// TwinCAT 3 PLC project MCSB
// ProgramVersion: 3.1.4024.0
// libraries:
//   Tc2_MC2, * (Beckhoff Automation GmbH)
//   Tc2_MC2_Drive, * (Beckhoff Automation GmbH)
//   Tc2_Standard, * (Beckhoff Automation GmbH)
//   Tc2_System, * (Beckhoff Automation GmbH)
//   Tc2_Utilities, * (Beckhoff Automation GmbH)
//   Tc3_Module, * (Beckhoff Automation GmbH)
// project tree:
//   DUTs/ ST_MC_CMD.TcDUT, ST_MC_Status.TcDUT
//   GVLs/ GVL.TcGVL
//   / PlcTask.TcTTO
//   POUs/ MAIN.TcPOU, MotionCtrl.TcPOU
// real-time tasks:
//   TASK PlcTask: cycle T#10ms, priority 20, ADS port 350
// motion (NC):
//   TASK NC-Task 1 SAF: cycle T#2ms, priority 4, ADS port 501
//   TASK NC-Task 1 SVB: cycle T#10ms, priority 8, ADS port 511
//   AXIS Axis 1 (id 1)
//     OtherSettings: AllowMotionCmdToSlave=true
//     encoder EncType=19
//       EncPara: MaxCount=#xffffffff
//     drive DrvType=16
//       DrvPara: MaxCount=#xffffffff
//         Analog: TorqueSetpointScale=10, ScaleFactorActTorque=0.1
//         TimeComp: TaskDelayCycles=1
//     controller CtrType=1
//       CtrPara: PriorControlFactor=1
//         Observer: BandWidth=20
//   AXIS Axis 2 (id 2)
//     Dynamic: Acceleration=1610, Deceleration=1610, Jerk=2124.67
//     OtherSettings: AllowMotionCmdToSlave=true
//     encoder EncType=7
//       EncPara: MaxCount=#x0000ffff, ReferenceSystem=1
//     drive DrvType=5
//       Analog: TorqueSetpointScale=10, ScaleFactorActTorque=0.1
//       TimeComp: TaskDelayCycles=1
//     controller CtrType=1
//       CtrPara: PriorControlFactor=1
//         Observer: BandWidth=20
//   AXIS Axis 3 Virtual (id 3)
//     OtherSettings: AllowMotionCmdToSlave=true
//     encoder EncType=1
//     drive DrvType=5
//       Analog: TorqueSetpointScale=10, ScaleFactorActTorque=0.1
//       TimeComp: TaskDelayCycles=1
//     controller CtrType=1
//       CtrPara: PriorControlFactor=1
//         Observer: BandWidth=20
// I/O:
//   DEVICE Device 1 (EtherCAT) (disabled), AmsNetId 10.0.2.15.2.1
//     Term 1 (EK1200) [EK1200-5000 EtherCAT Power supply (2A E-Bus)]
//       Term 2 (EL1008) [EL1008 8Ch. Dig. Input 24V, 3ms]
//       Term 3 (EL2008) [EL2008 8Ch. Dig. Output 24V, 0.5A]
//       Drive 4 (EL7201-0001) [EL7201-0001 1Ch. DS402 Servo motor output stage (50V, 4A)]
//       Term 5 (EL3042) [EL3042 2Ch. Ana. Input 0-20mA]
//       Term 6 (EL4012) [EL4012 2Ch. Ana. Output 0-20mA, 12bit]
//       Term 7 (EK1122) [EK1122 2 port EtherCAT junction]
// variable links:
//   MCSB/MCSB Instance <-> NC-Task 1 SAF/Axes/Axis 3 Virtual
//     PlcTask Inputs/GVL.SingleAxis.NcToPlc <-> Outputs/ToPlc
//     PlcTask Outputs/GVL.SingleAxis.PlcToNc <-> Inputs/FromPlc
//   (this object) <-> Device 1 (EtherCAT)/Term 1 (EK1200)/Drive 4 (EL7201-0001)
//     Drive/Inputs/In/nDcOutputTime <-> InfoData/DcOutputShift
//     Drive/Inputs/In/nState1 <-> DS402 Statusword/Statusword
//     Drive/Inputs/In/nState2 <-> DS402 Statusword/Statusword @bit 8
//     Drive/Inputs/In/nState4 @bit 1 <-> WcState/InputToggle
//     Drive/Inputs/In/nState4 <-> WcState/WcState
//     Drive/Outputs/Out/nCtrl1 <-> DS402 Controlword/Controlword
//     Drive/Outputs/Out/nCtrl2 <-> DS402 Controlword/Controlword @bit 8
//     Drive/Outputs/Out/nDataOut2 <-> DS402 Target velocity/Target velocity
//     Enc/Inputs/In/nDataIn1 <-> DS402 Position actual value/Position actual value
//     Enc/Inputs/In/nDcInputTime <-> InfoData/DcInputShift
//     Enc/Inputs/In/nState4 @bit 1 <-> WcState/InputToggle
//     Enc/Inputs/In/nState4 <-> WcState/WcState
//   (this object) <-> Device 1 (EtherCAT)/Term 1 (EK1200)/Term 5 (EL3042)
//     Enc/Inputs/In/nDataIn1[0] <-> AI Standard Channel 1/Value
//     Enc/Inputs/In/nState4 @bit 1 <-> WcState/InputToggle
//     Enc/Inputs/In/nState4 <-> WcState/WcState
//   (this object) <-> Device 1 (EtherCAT)/Term 1 (EK1200)/Term 6 (EL4012)
//     Drive/Inputs/In/nState4 <-> WcState/WcState
//     Drive/Outputs/Out/nDataOut1[0] <-> AO Outputs Channel 1/Analog output

CONFIGURATION MCSB
    RESOURCE PLC ON TwinCAT3
        TASK PlcTask(INTERVAL := T#10ms, PRIORITY := 20);
        PROGRAM MAIN WITH PlcTask : MAIN;
    END_RESOURCE
END_CONFIGURATION

// ---- DUTs/ST_MC_CMD.TcDUT
TYPE ST_MC_CMD :
STRUCT
	bExe	  		: BOOL;
	lrVelocity		: LREAL;
	lrAcceleration	: LREAL;
	lrDeceleration	: LREAL;
	lrJog			: LREAL;
	lrDistance		: LREAL;
	lrPosition		: LREAL;
	EnuDrecetion	: MC_Direction;
	EnuBufferMode	: MC_BufferMode;
	EnuOptions		: ST_MoveOptions;
END_STRUCT
END_TYPE

// ---- DUTs/ST_MC_Status.TcDUT
TYPE ST_MC_Status :
STRUCT
	Status	: BOOL;
	Done	: BOOL;
	Busy	: BOOL;
	Error	: BOOL;
	Active	: BOOL;
	CmdAborted	: BOOL;
	InVelocity	: BOOL;
	ErrorID	: UDINT;
	
END_STRUCT
END_TYPE

// ---- GVLs/GVL.TcGVL
{attribute 'qualified_only'}
VAR_GLOBAL
	SingleAxis : Axis_REF;
	
	
	fbSA_Reset 	: MC_RESET;
	fbSA_Power 	: MC_POWER;
	fbSA_Home 	: MC_HOME;
	fbSA_Jog 	: MC_JOG;
	fbSA_MovVel1 	: MC_MoveVelocity;
	fbSA_MovVel2 	: MC_MoveVelocity;
	fbSA_MovRel1 	: MC_MoveRelative;
	fbSA_MovRel2 	: MC_MoveRelative;
	fbSA_MoveAbs1 	: MC_MoveAbsolute;
	fbSA_MoveAbs2 	: MC_MoveAbsolute;
	
	bSA_ResetExe		: BOOL;
	
	bSA_PowerEnCmd		: BOOL;
	bSA_PowerEnPositive	: BOOL;
	bSA_PowerEnNegative	: BOOL;
	
	bSA_HomeExe			: BOOL;
	bSA_HomeCamInput	: BOOL;
	
	bSA_JogFwd			:BOOL;
	bSA_JogRev			:BOOL;
	
	stSA_VelCmd1			: ST_MC_CMD;
	stSA_VelCmd2			: ST_MC_CMD;
	stSA_RelCmd1			: ST_MC_CMD;
	stSA_RelCmd2			: ST_MC_CMD;
	stSA_AbsCmd1			: ST_MC_CMD;
	stSA_AbsCmd2			: ST_MC_CMD;
	
	
	iRSA_PowerOverride	: LREAL;
	iRSA_HomePosition	: LREAL;
	iRSA_SetPosition	: LREAL;
	iRSA_JogVelocity	: LREAL;
	
	stSA_Reset		: ST_MC_Status;
	stSA_Power		: ST_MC_Status;
	stSA_Home		: ST_MC_Status;
	stSA_SetPosition : ST_MC_Status;
	stSA_Jog		: ST_MC_Status;
	
	ST_VelSta1		: ST_MC_Status;
	ST_VelSta2		: ST_MC_Status;
	ST_RelSta1		: ST_MC_Status;
	ST_RelSta2		: ST_MC_Status;
	ST_AbsSta1		: ST_MC_Status;
	ST_AbsSta2		: ST_MC_Status;
	
	
END_VAR

// ---- POUs/MAIN.TcPOU
PROGRAM MAIN
VAR
END_VAR

MotionCtrl();

END_PROGRAM

// ---- POUs/MotionCtrl.TcPOU
PROGRAM MotionCtrl
VAR
END_VAR

SingleAxis_LD();

METHOD SingleAxis_LD : BOOL
VAR_INPUT
END_VAR
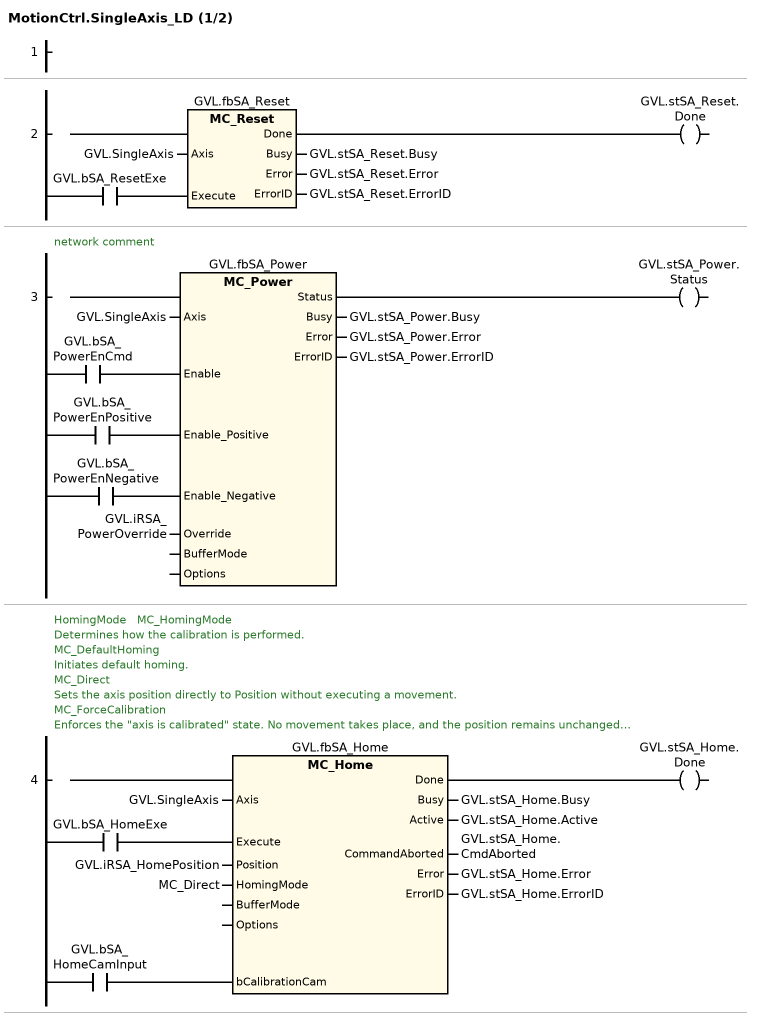
// NETWORK 1

// NETWORK 2
GVL.fbSA_Reset(
    Axis := GVL.SingleAxis,
    Execute := GVL.bSA_ResetExe,
    Busy => GVL.stSA_Reset.Busy,
    Error => GVL.stSA_Reset.Error,
    ErrorID => GVL.stSA_Reset.ErrorID); // MC_Reset
GVL.stSA_Reset.Done := GVL.fbSA_Reset.Done;

// NETWORK 3
// network comment
GVL.fbSA_Power(
    Axis := GVL.SingleAxis,
    Enable := GVL.bSA_PowerEnCmd,
    Enable_Positive := GVL.bSA_PowerEnPositive,
    Enable_Negative := GVL.bSA_PowerEnNegative,
    Override := GVL.iRSA_PowerOverride,
    Busy => GVL.stSA_Power.Busy,
    Error => GVL.stSA_Power.Error,
    ErrorID => GVL.stSA_Power.ErrorID); // MC_Power
GVL.stSA_Power.Status := GVL.fbSA_Power.Status;

// NETWORK 4
// HomingMode   MC_HomingMode
// Determines how the calibration is performed.
//
// MC_DefaultHoming
// Initiates default homing.
// MC_Direct
// Sets the axis position directly to Position without executing a movement.
// MC_ForceCalibration
// Enforces the "axis is calibrated" state. No movement takes place, and the position remains unchanged.
// MC_ResetCalibration
// Resets the calibration state of the axis. No movement takes place, and the position remains unchanged.
GVL.fbSA_Home(
    Axis := GVL.SingleAxis,
    Execute := GVL.bSA_HomeExe,
    Position := GVL.iRSA_HomePosition,
    HomingMode := MC_Direct,
    bCalibrationCam := GVL.bSA_HomeCamInput,
    Busy => GVL.stSA_Home.Busy,
    Active => GVL.stSA_Home.Active,
    CommandAborted => GVL.stSA_Home.CmdAborted,
    Error => GVL.stSA_Home.Error,
    ErrorID => GVL.stSA_Home.ErrorID); // MC_Home
GVL.stSA_Home.Done := GVL.fbSA_Home.Done;

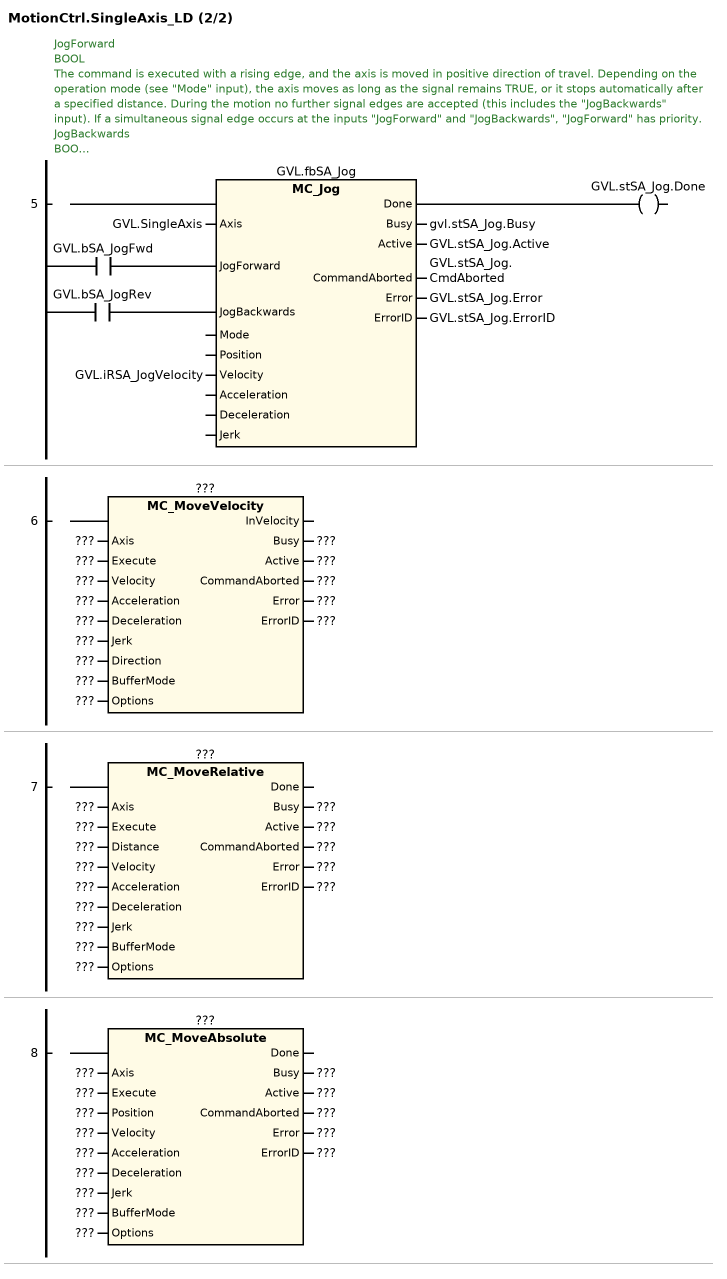
// NETWORK 5
// JogForward
//
// BOOL
//
// The command is executed with a rising edge, and the axis is moved in positive direction of travel. Depending on the operation mode (see "Mode" input), the axis moves as long as the signal remains TRUE, or it stops automatically after a specified distance. During the motion no further signal edges are accepted (this includes the "JogBackwards" input). If a simultaneous signal edge occurs at the inputs "JogForward" and "JogBackwards", "JogForward" has priority.
//
// JogBackwards
//
// BOOL
//
// The command is executed with a rising edge, and the axis is moved in negative direction of travel. "JogForward" and "JogBackwards" should be triggered alternatively, although they are also mutually locked internally.
//
// Mode
//
// E_JogMode
//
// Determines the operation mode in which the manual function is executed.
//
// MC_JOGMODE_STANDARD_SLOW
// the axis moves as long as the signal at one of the jog inputs is TRUE. The "low velocity for manual functions" specified in the TwinCAT System Manager and standard dynamics are used. In this operation mode the position, velocity and dynamics data specified in the function block have no effect.
// MC_JOGMODE_STANDARD_FAST
// the axis moves as long as the signal at one of the jog inputs is TRUE. The "high velocity for manual functions" specified in the TwinCAT System Manager and standard dynamics are used. In this operation mode the position, velocity and dynamics data specified in the function block have no effect.
// MC_JOGMODE_CONTINUOUS
// The axis moves as long as the signal at one of the jog inputs is TRUE. The velocity and dynamics data specified by the user are used. The position has no effect.
// MC_JOGMODE_INCHING
// With a rising edge at one of the jog inputs the axis is moved by a certain distance which is specified via the "Position" input. The axis stops automatically, irrespective of the state of the jog inputs. A new movement step is only executed once a further rising edge is encountered. With each start the velocity and dynamics data specified by the user are used.
// MC_JOGMODE_INCHING_MODULO
// With a rising edge at one of the jog inputs the axis is moved by a certain distance which is specified via the "Positions" input. The axis position will snap to an integer multiple of the position parameter. The axis stops automatically, irrespective of the state of the jog inputs. A new movement step is only executed once a further rising edge is encountered. With each start the velocity and dynamics data specified by the user are used.
// Position
//
// LREAL
//
// Relative distance for movements in MC_JOGMODE_INCHING operation mode.
//
// Velocity
//
// LREAL
//
// Maximum travel velocity (>0).
//
// Acceleration
//
// LREAL
//
// Acceleration (≥0). If the value is 0, the standard acceleration from the axis configuration in the System Manager is used.
//
// Deceleration
//
// LREAL
//
// Deceleration (≥0). If the value is 0, the standard deceleration from the axis configuration in the System Manager is used.
//
// Jerk
//
// LREAL
//
// Jerk (≥0). At a value of 0, the standard jerk from the axis configuration in the System Manager is applied.
GVL.fbSA_Jog(
    Axis := GVL.SingleAxis,
    JogForward := GVL.bSA_JogFwd,
    JogBackwards := GVL.bSA_JogRev,
    Velocity := GVL.iRSA_JogVelocity,
    Busy => gvl.stSA_Jog.Busy,
    Active => GVL.stSA_Jog.Active,
    CommandAborted => GVL.stSA_Jog.CmdAborted,
    Error => GVL.stSA_Jog.Error,
    ErrorID => GVL.stSA_Jog.ErrorID); // MC_Jog
GVL.stSA_Jog.Done := GVL.fbSA_Jog.Done;

// NETWORK 6
???(); // MC_MoveVelocity

// NETWORK 7
???(); // MC_MoveRelative

// NETWORK 8
???(); // MC_MoveAbsolute
END_METHOD

END_PROGRAM
